{attribute 'linkalways'} 
{attribute 'no_explicit_call' := 'This FB is a CLASS and must be accessed using methods or properties'}
{attribute 'enable_dynamic_creation'}
FUNCTION_BLOCK Node_F_VN_KeyPointsGFTT EXTENDS VisionNode
VAR
    ipSrcImage : _ITcVnImage;
    ipKeyPoints : _ITcVnContainer;
    hrPrev : _HRESULT(S_OK);
	hresult : _HRESULT(S_OK);
END_VAR

METHOD PUBLIC  Clone : I_Node
VAR
	pNode : POINTER TO Node_F_VN_KeyPointsGFTT;
END_VAR
pNode := __NEW(Node_F_VN_KeyPointsGFTT);
Clone := pNode^;
END_METHOD

METHOD FB_init : BOOL
VAR_INPUT
	bInitRetains : BOOL; // if TRUE, the retain variables are initialized (warm start / cold start)
	bInCopyCode : BOOL;  // if TRUE, the instance afterwards gets moved into the copy code (online change)
END_VAR
AddInput('ipSrcImage', ipSrcImage);
AddInput('hrPrev', hrPrev);
AddOutput('ipKeyPoints', ipKeyPoints);
AddOutput('hresult',hresult);
END_METHOD

METHOD PROTECTED OnExecute
hresult.Value := F_VN_KeyPointsGFTT(
	ipSrcImage := ipSrcImage.Value,
    ipKeyPoints := ipKeyPoints.Value,
	hrPrev:= hrPrev.Value);
END_METHOD

METHOD PUBLIC PreExecutionCheck
VAR_INPUT
	Check : I_PreExecutionChecks;
END_VAR
Check.IsTrue(ipSrcImage.IsValid, 'ipSrcImage must contain an image');
Check.IsTrue(ipSrcImage.HasChannelCount(1), 'ipSrcImage must have 1 channel');
END_METHOD

END_FUNCTION_BLOCK

(* stored: Version 1.1.0.1, ProductVersion 3.1.4024.15
   POU Node_F_VN_KeyPointsGFTT: Id {2e853095-783d-0c96-0bcd-4a103605683d}, SpecialFunc None
   Folder Constructor: Id {2bb24489-7827-03f9-38cf-7543040f5b24}
   Method Clone: Id {eb3cf41f-3390-09a5-2265-dab9b720f8ab}
   Method FB_init: Id {57bd5c52-bc1b-0d15-2d27-dedb110fbd84}
   Method OnExecute: Id {1ebdbc85-4d4f-0af2-1095-61ad84bef0b7}
   Method PreExecutionCheck: Id {2868df68-eb7a-052c-00e4-a6f4ff2020da} *)
